{attribute 'qualified_only'}
{attribute 'strict'}
TYPE DRIVE_STATE :
(
	SWITCH_ON_INHIBITED := 64,
	SWITCH_ON_INHIBITED_BIT_5 := 96,
	NOT_READY_TO_SWITCH_ON := 0,
	NOT_READY_TO_SWITCH_ON_BIT_5 := 32,
	READY_TO_SWITCH_ON := 33,
	SWITCHED_ON		   := 35,
	QUICK_STOP_ACTIVE	:= 7,
	OPERATION_ENABLED := 39,
	TROUBLE			:= 8,
	TROUBLE_BIT_5	:= 40,
	FAULT_REACTION_ACTIVE := 15,
	FAULT_REACTION_ACTIVE_BIT_5 := 47
) UINT;
END_TYPE

(* stored: Version 1.1.0.1, ProductVersion 3.1.4024.4
   EnumerationTextList DRIVE_STATE: Id {c80eb09b-c890-4023-9c6d-450875857e49} *)
